PROGRAM Manual
VAR
	Left:BOOL;
	Right:BOOL;
END_VAR

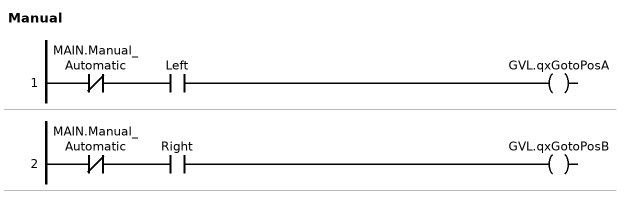
// NETWORK 1
GVL.qxGotoPosA := NOT MAIN.Manual_Automatic AND Left;

// NETWORK 2
GVL.qxGotoPosB := NOT MAIN.Manual_Automatic AND Right;

END_PROGRAM

(* stored: Version 1.1.0.1, ProductVersion 3.1.4024.12
   POU Manual: Id {827848a0-53f1-4e41-acf9-8f6a40ff5592}, SpecialFunc None *)
